TYPE ST_PowerGroupOutCmd :
STRUCT
    PowerOn : BOOL;
END_STRUCT
END_TYPE

(* stored: Version 1.1.0.1, ProductVersion 3.1.4024.12
   DUT ST_PowerGroupOutCmd: Id {de1a73e2-8ac7-4309-a1d6-202a8bd7b74f} *)
